# EPICS substitutions: ioc/bsread.subs
file bsread.template {
    {
        P="BSREAD"
    }
}
